{attribute addProperty BoxType "EL3356-0030-0025"}
{attribute addProperty Id "StatusAT %I*Status_F881FBAF162"}
{attribute addProperty CRC "2138159664"}
{attribute addProperty SizeInBites "16"}
{attribute addProperty SizeInBytes "2"}
TYPE RMB_Status_7F71BA30 :
STRUCT
	{attribute addProperty Name "Status"}
	Status AT %I* : Status_F881FBAF;
END_STRUCT
END_TYPE

(* stored: Version 1.2.0.0, ProductVersion 3.1.4024.9
   DUT RMB_Status_7F71BA30: Id {8897cdfc-26ed-4cdf-a8f6-5de81b7545c4} *)
